(* PLC project Laboratorio2, Desconocido Sin nombre 1 *)
(* stored: creationDateTime 2024-10-31T18:16:06, modificationDateTime 2024-11-03T23:48:20 *)

PROGRAM PLC_PRG
  VAR
    Sensor_X AT %IX0.0 : BOOL;
    Sensor_Y AT %IX0.1 : BOOL;
    LED_Amarillo AT %QX0.0 : BOOL;
    LED_Rojo AT %QX0.1 : BOOL;
  END_VAR
  VAR
    TON0 : TON;
    TON2 : TON;
  END_VAR

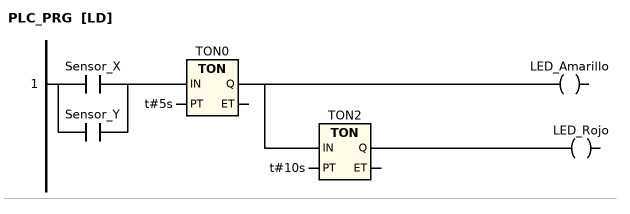
(* LD diagram, written out as Structured Text *)
TON0(IN := Sensor_X OR Sensor_Y, PT := t#5s);
LED_Amarillo := TON0.Q;
TON2(IN := TON0.Q, PT := t#10s);
LED_Rojo := TON2.Q;
END_PROGRAM

CONFIGURATION Config0
  RESOURCE Res0 ON PLC
    TASK task0(INTERVAL := T#20ms, PRIORITY := 0);
    PROGRAM instance0 WITH task0 : PLC_PRG;
  END_RESOURCE
END_CONFIGURATION
